FUNCTION_BLOCK OneUPS
VAR_INPUT
	Crit_Alm : BOOL;
	Minor_Alm : BOOL;
	ByPass_Mode : BOOL;
	Batt_Mode : BOOL;
	Offline : BOOL;
END_VAR
VAR_OUTPUT
END_VAR
VAR_TEMP
	 i : INT;
END_VAR

i := GVL.nInputCoilIndex;

GVL.mb_Input_Coils[i+0] := Crit_Alm;
GVL.mb_Input_Coils[i+1] := Minor_Alm;
GVL.mb_Input_Coils[i+2] := ByPass_Mode;
GVL.mb_Input_Coils[i+3] := Batt_Mode;
GVL.mb_Input_Coils[i+4] := Offline;

GVL.nInputCoilIndex := i + 5;

END_FUNCTION_BLOCK

(* stored: Version 1.1.0.1, ProductVersion 3.1.4024.12
   POU OneUPS: Id {eb4b6242-8091-4738-9c7d-0a3305c0ad6e}, SpecialFunc None *)
